{attribute 'qualified_only'}
{attribute 'strict'}
TYPE OrderToteErrorStatus:
(
	UNKNOWN							:=0,
  	NO_ERROR						:=1,
	MACHINE_NOT_RUNNING				:=2,
	ELECTRICAL_ERROR				:=3,
 	MECHANICAL_ERROR				:=4,
 	SAFETY_ERROR					:=5,
	UPSTREAM_NOT_READY				:=6,
	TIMEOUT_WAITING_FOR_NEW_TOTE	:=7,
	DOWNSTREAM_NOT_READY			:=8,
	TIMEOUT_WAITING_FOR_SPACE		:=9
);
END_TYPE

(* stored: Version 1.1.0.1, ProductVersion 3.1.4024.12
   DUT OrderToteErrorStatus: Id {91b4f0cf-44a7-448b-adb3-171992671f23} *)
